TYPE ST_Tank :
STRUCT
	 nId : INT;
     rtemperature : REAL;   // current temperature in celsius   
     rlevel : REAL;         // current fill level in percentage
     bAlarm : BOOL ;
END_STRUCT
END_TYPE

(* stored: Version 1.1.0.1, ProductVersion 3.1.4024.16
   DUT ST_Tank: Id {ed9b2ace-c862-4453-a289-3e174366ea4a} *)
